RoboDK station: EJRobot.rdk

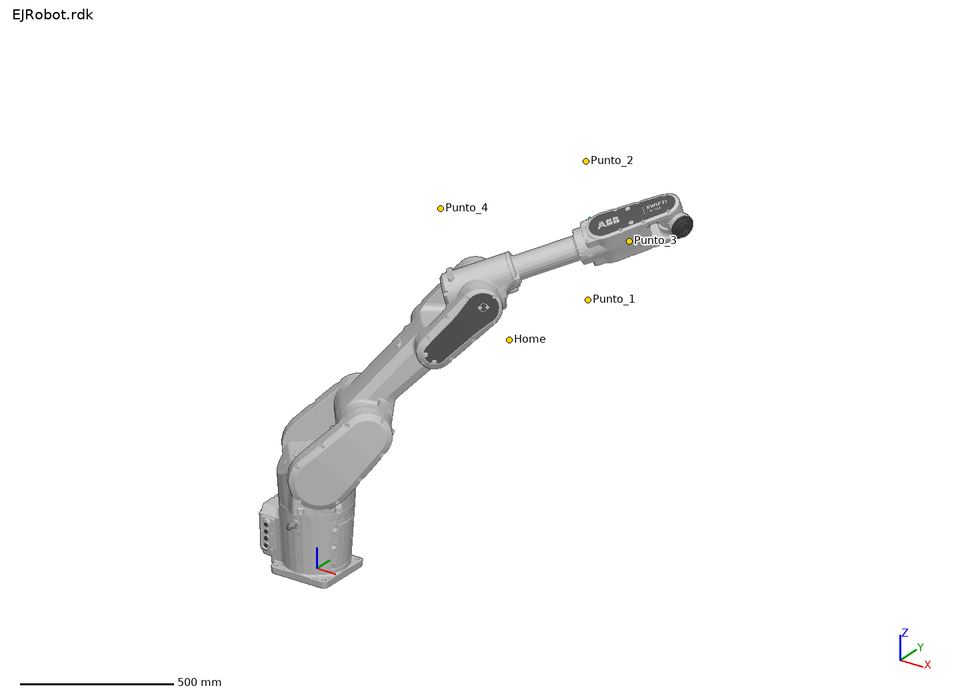
[picture v0: the station drawn from its stored meshes, robots at their saved joint values, targets as dots, program paths as lines]
Station EJRobot (saved by RoboDK 6.0.4). Poses are relative to the parent item; angles as X-Y-Z fixed-axis rotations.
  - frame ABB CRB 1300-7/1.4 Base at (0, 0, 0) mm
    - robot ABB CRB 1300-7/1.4: 6 axes
        modified DH rows (alpha deg, a mm, theta deg, d mm): 0, 0, 0, 544; -90, 150, -90, 0; 0, 575, 0, 0; -90, 40, 0, 675; 90, 0, 0, 0; -90, 0, 180, 90
        joint limits [-180, -95, -210, -230, -130, -242] to [180, 155, 69, 230, 130, 242]; home [0, 0, 0, 0, 0, 0]; saved at [39.343, 40.741, -59.35, -71.017, 64.165, 49.852]
    - target Home (Cartesian target) at (974.9, -299.89, 1220.5) mm, rotated rx -118.44 ry 73.1 rz -137.29 deg; joints [-16.83, 11.7, -19.04, -11.39, 15.6, -3.55] of ABB CRB 1300-7/1.4
    - target Punto_1 (Cartesian target) at (1016.23, 87.33, 1220.5) mm, rotated rx -118.44 ry 73.1 rz -115.28 deg; joints [5.18, 11.7, -19.04, -11.39, 15.6, -3.55] of ABB CRB 1300-7/1.4
    - target Punto_3 (Cartesian target) at (876.02, 522.45, 1220.5) mm, rotated rx -118.44 ry 73.1 rz -89.38 deg; joints [31.08, 11.7, -19.04, -11.39, 15.6, -3.55] of ABB CRB 1300-7/1.4
    - target Punto_2 (Cartesian target) at (418.58, 930.13, 1220.5) mm, rotated rx -118.44 ry 73.1 rz -54.42 deg; joints [66.04, 11.7, -19.04, -11.39, 15.6, -3.55] of ABB CRB 1300-7/1.4
    - target Punto_4 (Cartesian target) at (-339.94, 1188, 733.27) mm, rotated rx -158.3 ry 50.88 rz -50.41 deg; joints [106.19, 39.68, -19.04, -11.39, 15.6, -3.55] of ABB CRB 1300-7/1.4
  - Python program Main (listed below)

--- Python program Main ---
# Type help("robodk.robolink") or help("robodk.robomath") for more information
# Press F5 to run the script
# Documentation: https://robodk.com/doc/en/RoboDK-API.html
# Reference:     https://robodk.com/doc/en/PythonAPI/robodk.html
# Note: It is not required to keep a copy of this file, your Python script is saved with your RDK project

# You can also use the new version of the API:
from robodk import robolink    # RoboDK API
from robodk import robomath    # Robot toolbox


rlink = robolink.Robolink()    # RoboDK API

robot = rlink.Item("", robolink.ITEM_TYPE_ROBOT)

vHome = rlink.Item('Home')  # Home position (must be defined in the station)
vPunto_1 = rlink.Item('Punto_1')  # Target 1 (must be defined in the station)
vPunto_2 = rlink.Item('Punto_2')  # Target
vPunto_3 = rlink.Item('Punto_3')  # Target 3 (must be defined in the station)
vPunto_4 = rlink.Item('Punto_4')  # Target 4 (must be defined in the station)

robot.MoveJ(vHome)  # Move to the home position
robot.MoveJ(vPunto_1)  # Move to target 1
robot.MoveJ(vPunto_2)  # Move to target 2
robot.MoveJ(vPunto_3)  # Move to target 3
robot.MoveJ(vPunto_4)  # Move to target 4
